// Mitsubishi GX Works2 project: PLC_GROUP11   PLC: FX3G

// global labels: Global1
VAR_GLOBAL
  start_day AT X007 : BOOL;
  yeast_input AT D1100 : REAL;
  yeast AT D1102 : REAL;
  end_day AT M100 : BOOL;
  malt_input AT D1104 : REAL;
  malt AT D1106 : REAL;
  fluff_input AT D1108 : REAL;
  fluff AT D1110 : REAL;
  work_day AT Y007 : BOOL;
  emergency AT X011 : BOOL;
  start_brew AT X001 : BOOL;
  timer_brew_4 AT TC1 : BOOL;
END_VAR
VAR_GLOBAL CONSTANT
  four_sec_brew : INT := 40;
END_VAR
VAR_GLOBAL
  is_brewing AT Y001 : BOOL;
END_VAR
VAR_GLOBAL CONSTANT
  five : INT := 2020;
END_VAR
VAR_GLOBAL
  lager AT M0 : BOOL;
  pilzner AT M2 : BOOL;
  analog_1_val AT D2000 : INT;
  analog1 AT D8280 : INT;
  start_ferment AT X005 : BOOL;
  timer_fermen_pilzner AT TC3 : BOOL;
  timer_ferment_lager AT TC2 : BOOL;
  timer_ferm_2 AT TC4 : BOOL;
  timer_ferm_1 AT TC5 : BOOL;
  lamp4 AT Y004 : BOOL;
  lamp3 AT Y003 : BOOL;
  timer_brew_finish AT TS1 : BOOL;
  ferment_cycle AT M11 : BOOL;
  timer_ferm_2_finish AT TS4 : BOOL;
  timer_ferm_1_finish AT TS5 : BOOL;
  timer_ferment_lager_finish AT TS2 : BOOL;
  timer_ferment_pilsner_finish AT TS3 : BOOL;
  ferment_finish AT M20 : BOOL;
  start_storage AT X002 : BOOL;
  pack_bottle AT X000 : BOOL;
  counter_packing AT CC1 : BOOL;
  bottles_packed AT CN1 : INT;
  new_pack AT M30 : BOOL;
  lamp2 AT Y002 : BOOL;
  counter_packing_finished AT CS1 : BOOL;
END_VAR
VAR_GLOBAL CONSTANT
  sub_120 : REAL := 120;
  sub_150 : REAL := 150;
  sub_12 : REAL := 12;
  sub_60 : REAL := 60;
  sub_6 : REAL := 6;
  sub_53 : REAL := 53;
END_VAR
VAR_GLOBAL
  brew_finish AT M22 : BOOL;
  packing_finish AT M24 : BOOL;
  storage AT D3000 : INT;
  analog_output AT D8282 : INT;
END_VAR
VAR_GLOBAL CONSTANT
  pilzner_min_yeast : REAL := 120;
  pilzner_min_malt : REAL := 6;
  pilzner_min_fluff : REAL := 53;
  lager_min_yeast : REAL := 150;
  lager_min_malt : REAL := 12;
  lager_min_fluff : REAL := 60;
END_VAR
VAR_GLOBAL
  cannot_brew_error AT M97 : BOOL;
  material_empty AT M98 : BOOL;
END_VAR
VAR_GLOBAL CONSTANT
  zero : INT;
  three_sec : INT := 30;
  four_sec : INT := 40;
  blink_const : INT := 5;
  six_bottles : INT := 6;
  one_to_storge : INT := 1;
  divider_ten : INT := 10;
  mul_404 : INT := 404;
END_VAR

// task Task_01 (event TRUE, interval 0, priority 31): POU_01

PROGRAM POU_01
(* structured ladder/FBD written out as ST: instructions are called as NAME(EN, inputs, outputs); _pN, _eN, _tN stand for wires *)
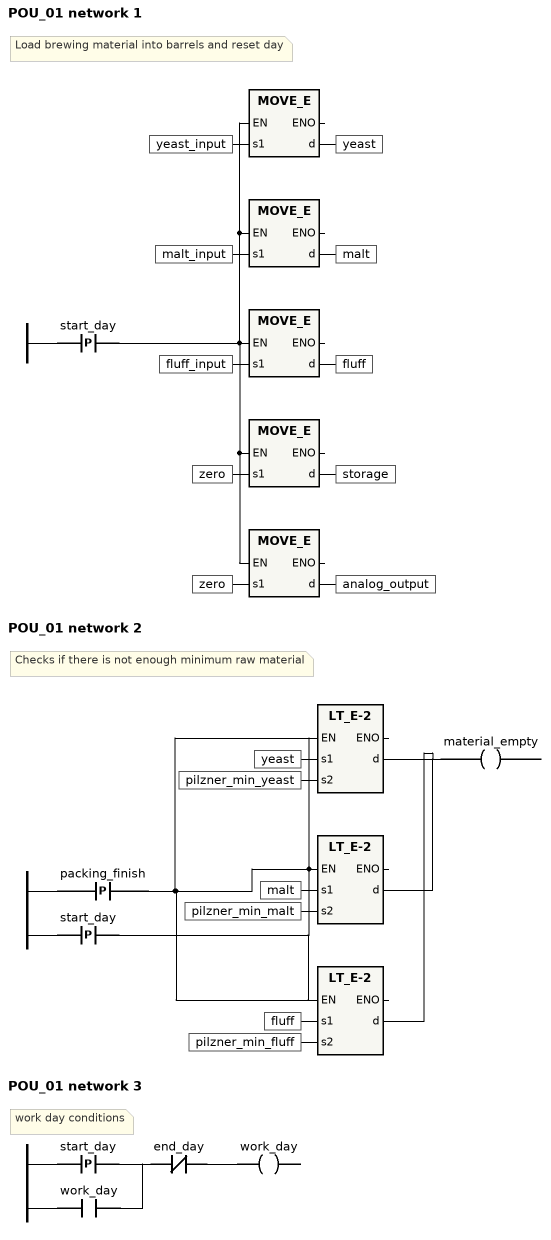
(* network 1 *)
(* Load brewing material into barrels and reset day *)
_p1 := LDP(TRUE, start_day);
MOVE_E(_p1, yeast_input, yeast);
MOVE_E(_p1, malt_input, malt);
MOVE_E(_p1, fluff_input, fluff);
MOVE_E(_p1, zero, storage);
MOVE_E(_p1, zero, analog_output);
(* network 2 *)
(* Checks if there is not enough minimum raw material *)
_p1 := LDP(TRUE, packing_finish) OR LDP(TRUE, start_day);
LT_E(_p1, yeast, pilzner_min_yeast, _t2);
LT_E(_p1, malt, pilzner_min_malt, _t3);
LT_E(_p1, fluff, pilzner_min_fluff, _t4);
material_empty := _t2 OR _t3 OR _t4;
(* network 3 *)
(* work day conditions *)
work_day := (LDP(TRUE, start_day) OR work_day) AND NOT end_day;
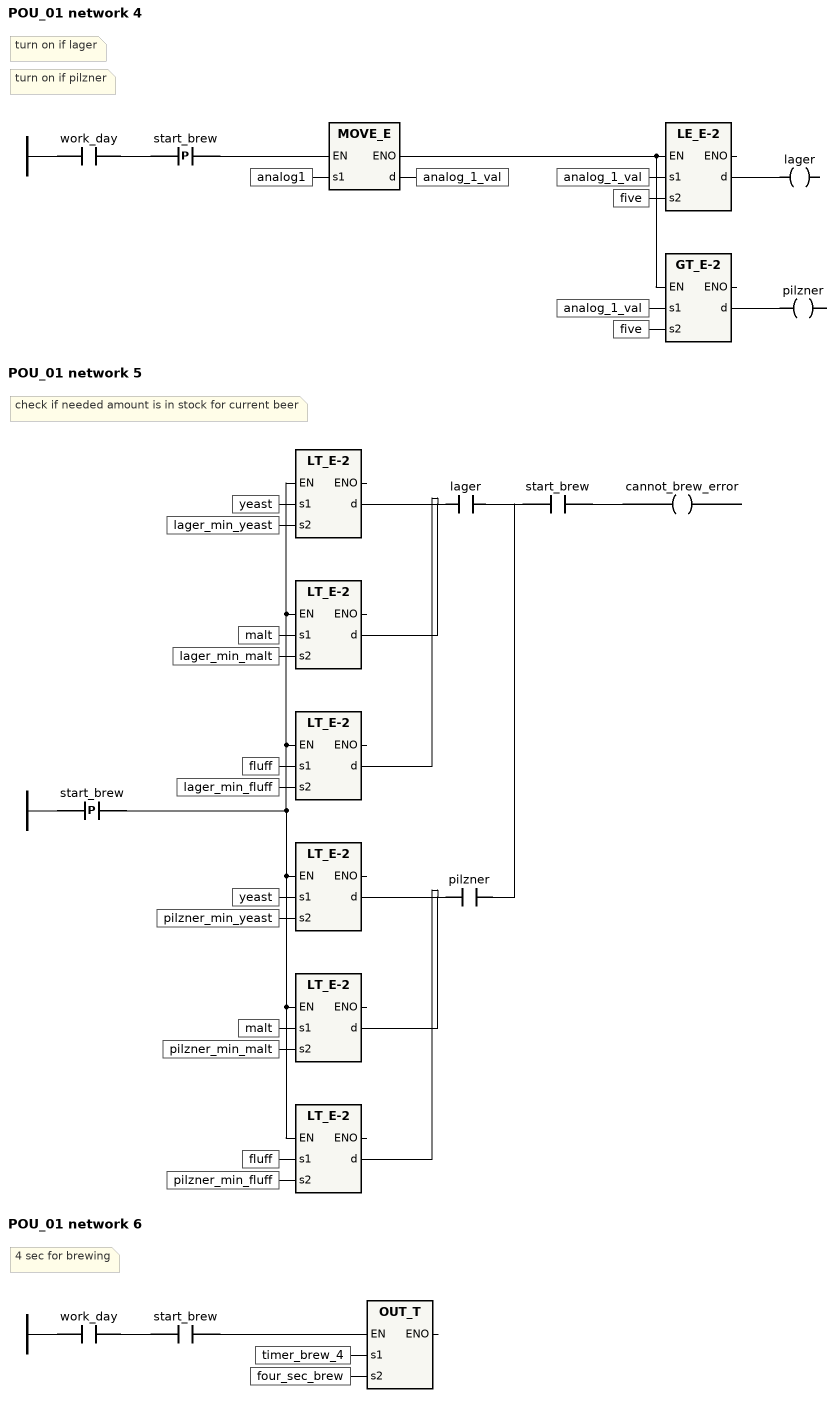
(* network 4 *)
(* turn on if lager *)
(* turn on if pilzner *)
_e1 := MOVE_E(work_day AND LDP(TRUE, start_brew), analog1, analog_1_val);
LE_E(_e1, analog_1_val, five, _t2);
lager := _t2;
GT_E(_e1, analog_1_val, five, _t3);
pilzner := _t3;
(* network 5 *)
(* check if needed amount is in stock for current beer *)
_p1 := LDP(TRUE, start_brew);
LT_E(_p1, yeast, lager_min_yeast, _t2);
LT_E(_p1, malt, lager_min_malt, _t3);
LT_E(_p1, fluff, lager_min_fluff, _t4);
LT_E(_p1, yeast, pilzner_min_yeast, _t5);
LT_E(_p1, malt, pilzner_min_malt, _t6);
LT_E(_p1, fluff, pilzner_min_fluff, _t7);
cannot_brew_error := (((_t2 OR _t3 OR _t4) AND lager) OR ((_t5 OR _t6 OR _t7) AND pilzner)) AND start_brew;
(* network 6 *)
(* 4 sec for brewing *)
OUT_T(work_day AND start_brew, timer_brew_4, four_sec_brew);
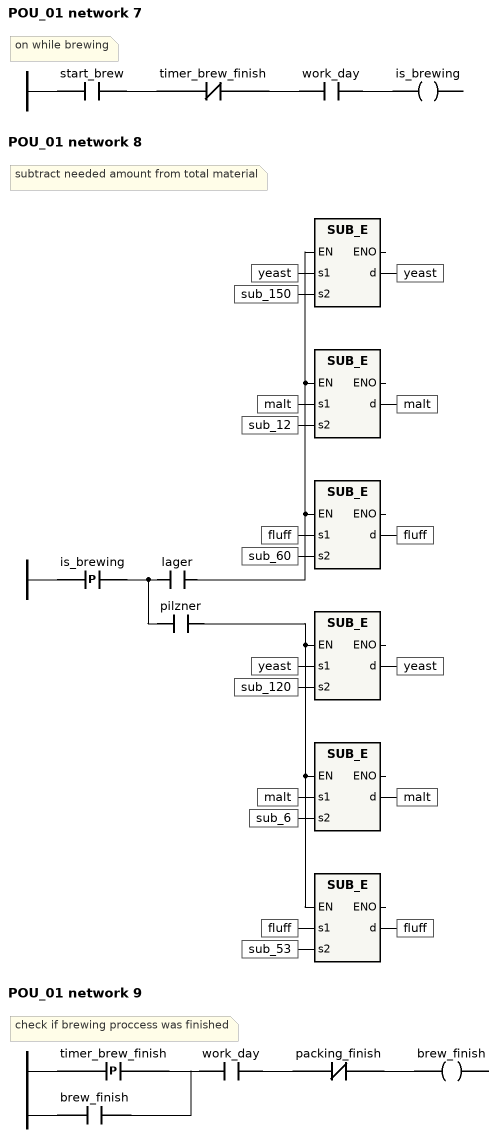
(* network 7 *)
(* on while brewing *)
is_brewing := start_brew AND NOT timer_brew_finish AND work_day;
(* network 8 *)
(* subtract needed amount from total material *)
_p1 := LDP(TRUE, is_brewing);
_p2 := _p1 AND lager;
SUB_E(_p2, yeast, sub_150, yeast);
SUB_E(_p2, malt, sub_12, malt);
SUB_E(_p2, fluff, sub_60, fluff);
_p3 := _p1 AND pilzner;
SUB_E(_p3, yeast, sub_120, yeast);
SUB_E(_p3, malt, sub_6, malt);
SUB_E(_p3, fluff, sub_53, fluff);
(* network 9 *)
(* check if brewing proccess was finished *)
brew_finish := ((LDP(TRUE, timer_brew_finish) OR brew_finish) AND work_day) AND NOT packing_finish;
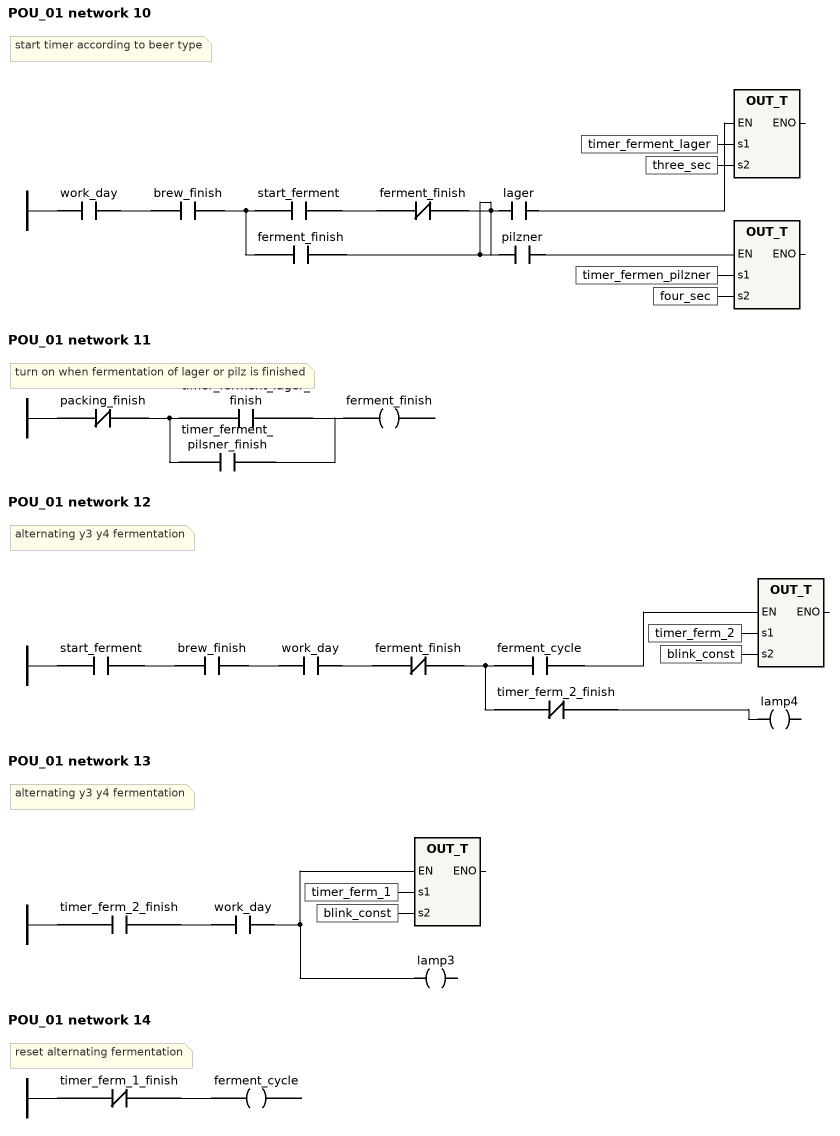
(* network 10 *)
(* start timer according to beer type *)
_p1 := work_day AND brew_finish;
_p2 := (_p1 AND start_ferment AND NOT ferment_finish) OR (_p1 AND ferment_finish);
OUT_T(_p2 AND lager, timer_ferment_lager, three_sec);
OUT_T(_p2 AND pilzner, timer_fermen_pilzner, four_sec);
(* network 11 *)
(* turn on when fermentation of lager or pilz is finished *)
_p1 := NOT packing_finish;
ferment_finish := (_p1 AND timer_ferment_lager_finish) OR (_p1 AND timer_ferment_pilsner_finish);
(* network 12 *)
(* alternating y3 y4 fermentation *)
_p1 := start_ferment AND brew_finish AND work_day AND NOT ferment_finish;
OUT_T(_p1 AND ferment_cycle, timer_ferm_2, blink_const);
lamp4 := _p1 AND NOT timer_ferm_2_finish;
(* network 13 *)
(* alternating y3 y4 fermentation *)
_p1 := timer_ferm_2_finish AND work_day;
OUT_T(_p1, timer_ferm_1, blink_const);
lamp3 := _p1;
(* network 14 *)
(* reset alternating fermentation *)
ferment_cycle := NOT timer_ferm_1_finish;
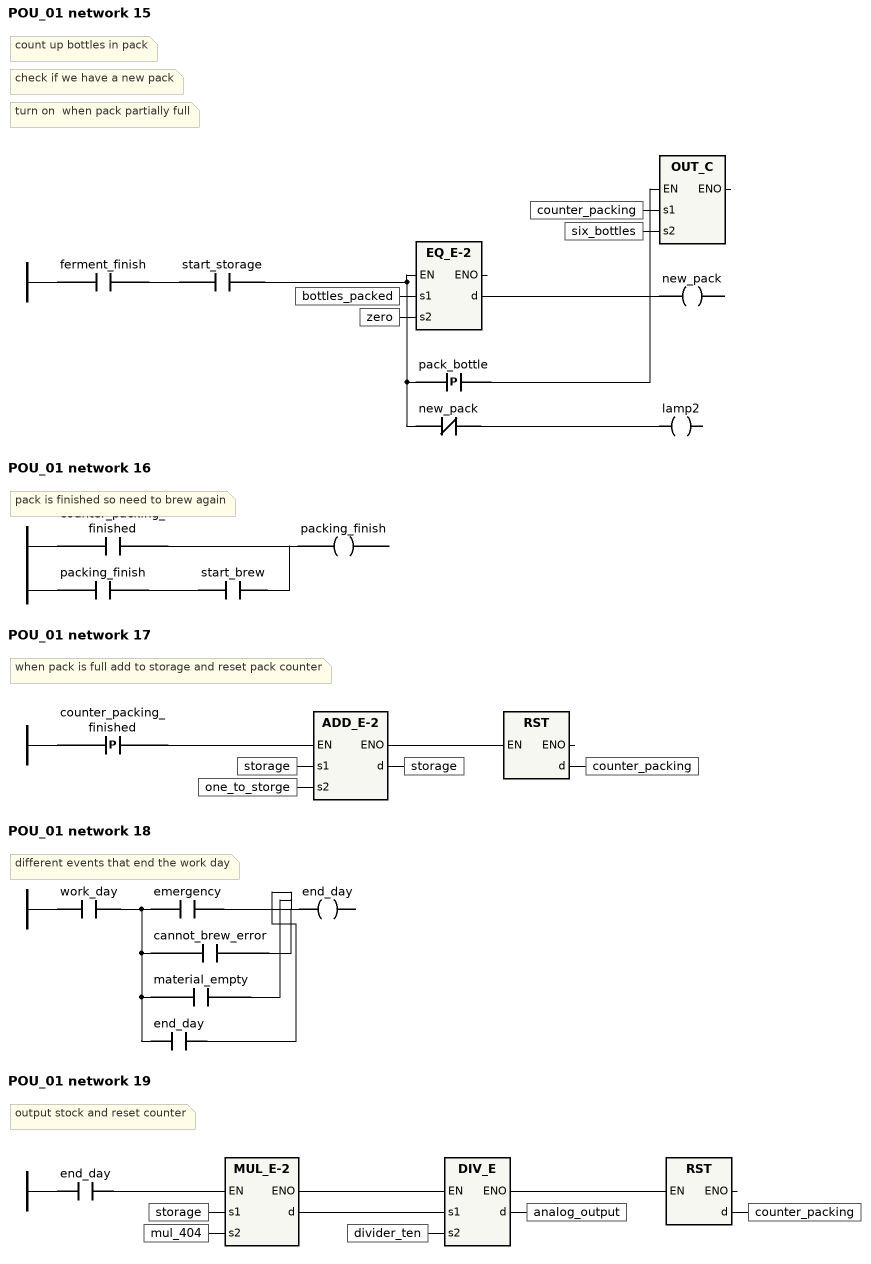
(* network 15 *)
(* count up bottles in pack *)
(* check if we have a new pack *)
(* turn on  when pack partially full *)
_p1 := ferment_finish AND start_storage;
OUT_C(_p1 AND LDP(TRUE, pack_bottle), counter_packing, six_bottles);
EQ_E(_p1, bottles_packed, zero, _t2);
new_pack := _t2;
lamp2 := _p1 AND NOT new_pack;
(* network 16 *)
(* pack is finished so need to brew again *)
packing_finish := counter_packing_finished OR (packing_finish AND start_brew);
(* network 17 *)
(* when pack is full add to storage and reset pack counter *)
_e1 := ADD_E(LDP(TRUE, counter_packing_finished), storage, one_to_storge, storage);
RST(_e1, counter_packing);
(* network 18 *)
(* different events that end the work day *)
end_day := (work_day AND emergency) OR (work_day AND cannot_brew_error) OR (work_day AND material_empty) OR (work_day AND end_day);
(* network 19 *)
(* output stock and reset counter *)
_e2 := MUL_E(end_day, storage, mul_404, _t1);
_e3 := DIV_E(_e2, _t1, divider_ten, analog_output);
RST(_e3, counter_packing);
END_PROGRAM
